(* Schneider Machine Expert - Basic project PICK AND PLACE 1.2mantep, file version 2.7.0.0 *)
(* ProjectInformations: Name=New project *)

HARDWARE
  Cpu 0: TM221CE40R
  EthernetConfiguration: NetworkName=M221, IpAllocationMode=FixedAddress, IpAddress=192.168.0.12, SubnetMask=255.255.255.0
  SerialLineConfiguration: Baud=Baud19200, Parity=ParityEven, DataBits=DataBits8, StopBits=StopBits1, PhysicalMedium=PhysicalMediumRs485, TransmissionMode=TransmissionModeModbusRtu, SlaveId=1, Addressing=SlaveAddressing
  MastTask: UsePeriodScanMode=false, PeriodScan=100
  FastTask: Period=255
  CpuBehavior: StartingMode=StartAsPreviousState, AutoSaveRamOnEeprom=true, WatchdogPeriod=250

SYMBOLS  (address, symbol, comment, settings)
  %M0         "K EMG"
  %M1         "K RESET"
  %M2         "RESET CLEAR"
  %M10        "K AUTO"
  %M11        "K1"
  %M12        "K2"
  %M13        "K3"
  %M14        "K4"
  %M15        "K CYC"
  %M16        "K STOP"
  %M17        "K5"
  %M50        "STEP"
  %M51        "K1 STEP"
  %M52        "K2 STEP"
  %M53        "K3 STEP"
  %M54        "K4 STEP"
  %M57        "K5 STEP"
  %M100       "kAmin"
  %M101       "kAplus"
  %M102       "kBmin"
  %M103       "kBplus"
  %M104       "kVakum"
  %M105       "KLHijau"
  %M106       "kLMerah"
  %M107       "kLKuning"
  %M200       "kB1"
  %M201       "kStart"
  %M202       "kStop"
  %M203       "kReset"
  %M204       "kA/S"
  %M205       "kS/C"
  %M206       "kA0"
  %M207       "kLimitS"
  %M208       "kProxy"
  %M209       "kB1min"
  %M210       "kVakum"
  %M211       "kBplus"
  %M212       "kAmin"
  %M213       "kBmin"
  %M214       "kAplus"
  %M215       "kLrun"
  %M216       "kLstop"
  %M217       "kLReset"
  %M400       "M.koilStart"
  %M500       "M.Start"
  %M501       "M.stop"
  %M510       "Mmasterstart"
  %M511       "R_Trig"
  %M700       "K.start"
  %TM0        [Preset=1, Base=OneSecond]
  %TM1        [Preset=1, Base=OneSecond]
  %I0.0       "EMG"
  %I0.1       "START"
  %I0.2       "STOP"
  %I0.3       "RESET"
  %I0.4       "AUTO/STEP"
  %I0.5       "SGL/CYC"
  %I0.7       "A1"
  %I0.10      "A0"
  %I0.11      "LS"
  %I0.12      "PROXY"
  %I0.13      "B1"
  %I0.14      "B1"
  %Q0.3       "VAKUUM"
  %Q0.4       "B+"
  %Q0.5       "A-"
  %Q0.6       "B-"
  %Q0.7       "A+"
  %Q0.11      "IND RUN"
  %Q0.12      "IND STOP"
  %Q0.15      "IND RESET"

POU EMG
  (* SectionNumber=1 *)

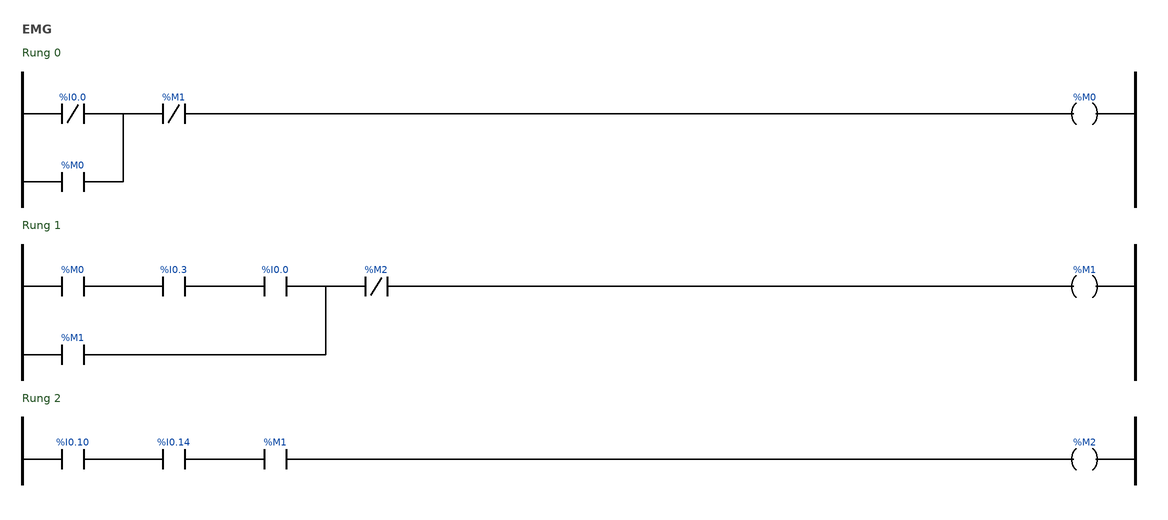

// Rung 0
  LDN %I0.0
  OR %M0
  ANDN %M1
  ST %M0
  // as ST:
  //   %M0 := (NOT %I0.0 OR %M0) AND NOT %M1;

// Rung 1
  LD %M0
  AND %I0.3
  AND %I0.0
  OR %M1
  ANDN %M2
  ST %M1
  // as ST:
  //   %M1 := (%M0 AND %I0.3 AND %I0.0 OR %M1) AND NOT %M2;

// Rung 2
  LD %I0.10
  AND %I0.14
  AND %M1
  ST %M2
  // as ST:
  //   %M2 := %I0.10 AND %I0.14 AND %M1;

POU OUTPUT
  (* SectionNumber=2 *)

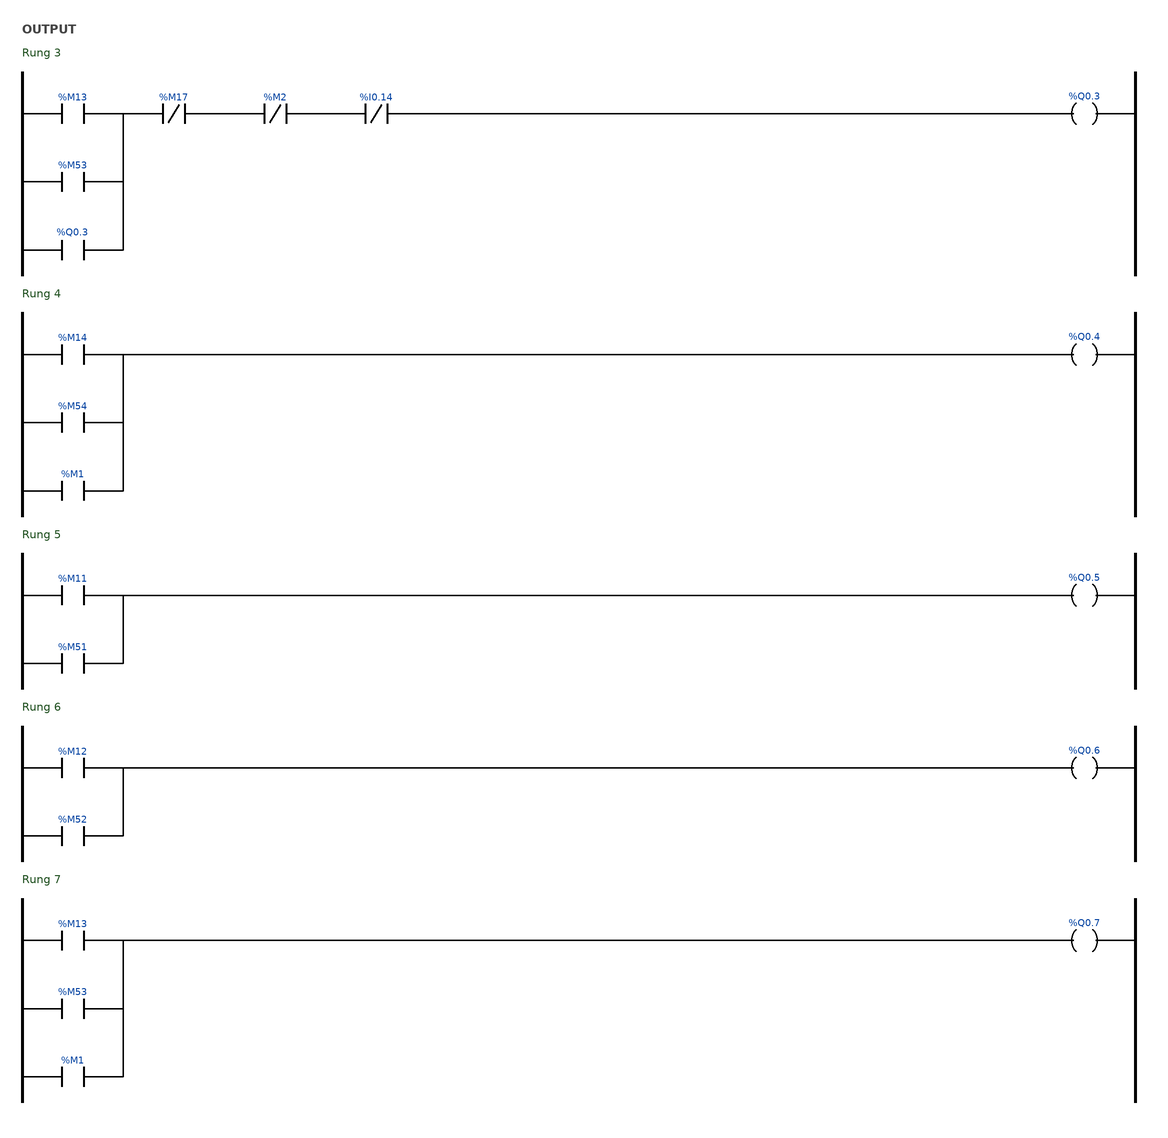

// Rung 3
  LD %M13
  OR %M53
  OR %Q0.3
  ANDN %M17
  ANDN %M2
  ANDN %I0.14
  ST %Q0.3
  // as ST:
  //   %Q0.3 := (%M13 OR %M53 OR %Q0.3) AND NOT %M17 AND NOT %M2 AND NOT %I0.14;

// Rung 4
  LD %M14
  OR %M54
  OR %M1
  ST %Q0.4
  // as ST:
  //   %Q0.4 := %M14 OR %M54 OR %M1;

// Rung 5
  LD %M11
  OR %M51
  ST %Q0.5
  // as ST:
  //   %Q0.5 := %M11 OR %M51;

// Rung 6
  LD %M12
  OR %M52
  ST %Q0.6
  // as ST:
  //   %Q0.6 := %M12 OR %M52;

// Rung 7
  LD %M13
  OR %M53
  OR %M1
  ST %Q0.7
  // as ST:
  //   %Q0.7 := %M13 OR %M53 OR %M1;

POU AUTO
  (* SectionNumber=3 *)

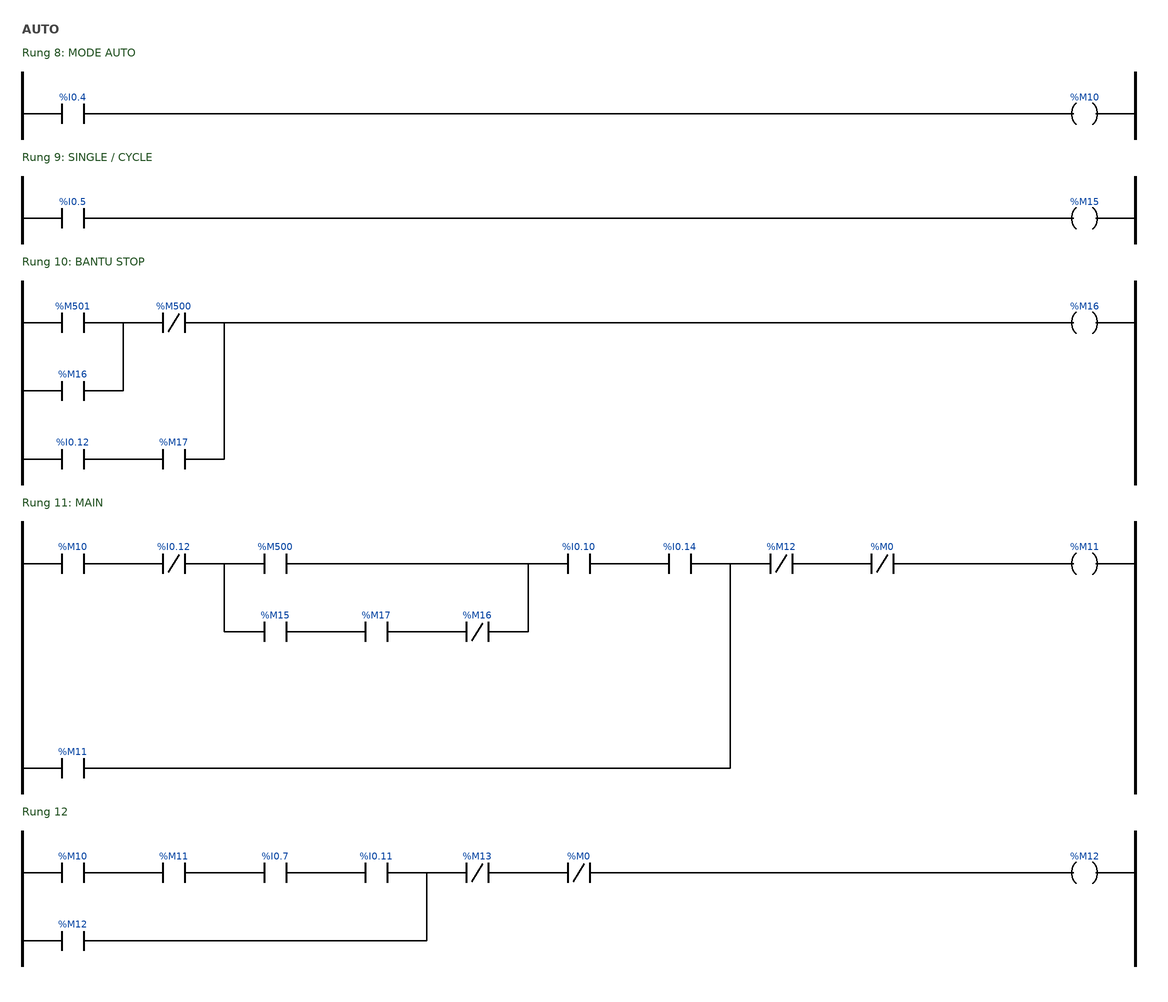

// Rung 8: MODE AUTO
  LD %I0.4
  ST %M10
  // as ST:
  //   %M10 := %I0.4;

// Rung 9: SINGLE / CYCLE
  LD %I0.5
  ST %M15
  // as ST:
  //   %M15 := %I0.5;

// Rung 10: BANTU STOP
  LD %M501
  OR %M16
  ANDN %M500
  OR( %I0.12
  AND %M17
  )
  ST %M16
  // as ST:
  //   %M16 := (%M501 OR %M16) AND NOT %M500 OR %I0.12 AND %M17;

// Rung 11: MAIN
  LD %M10
  ANDN %I0.12
  AND( %M500
  OR( %M15
  AND %M17
  ANDN %M16
  )
  )
  AND %I0.10
  AND %I0.14
  OR %M11
  ANDN %M12
  ANDN %M0
  ST %M11
  // as ST:
  //   %M11 := (%M10 AND NOT %I0.12 AND (%M500 OR %M15 AND %M17 AND NOT %M16) AND %I0.10 AND %I0.14 OR %M11) AND NOT %M12 AND NOT %M0;

// Rung 12
  LD %M10
  AND %M11
  AND %I0.7
  AND %I0.11
  OR %M12
  ANDN %M13
  ANDN %M0
  ST %M12
  // as ST:
  //   %M12 := (%M10 AND %M11 AND %I0.7 AND %I0.11 OR %M12) AND NOT %M13 AND NOT %M0;

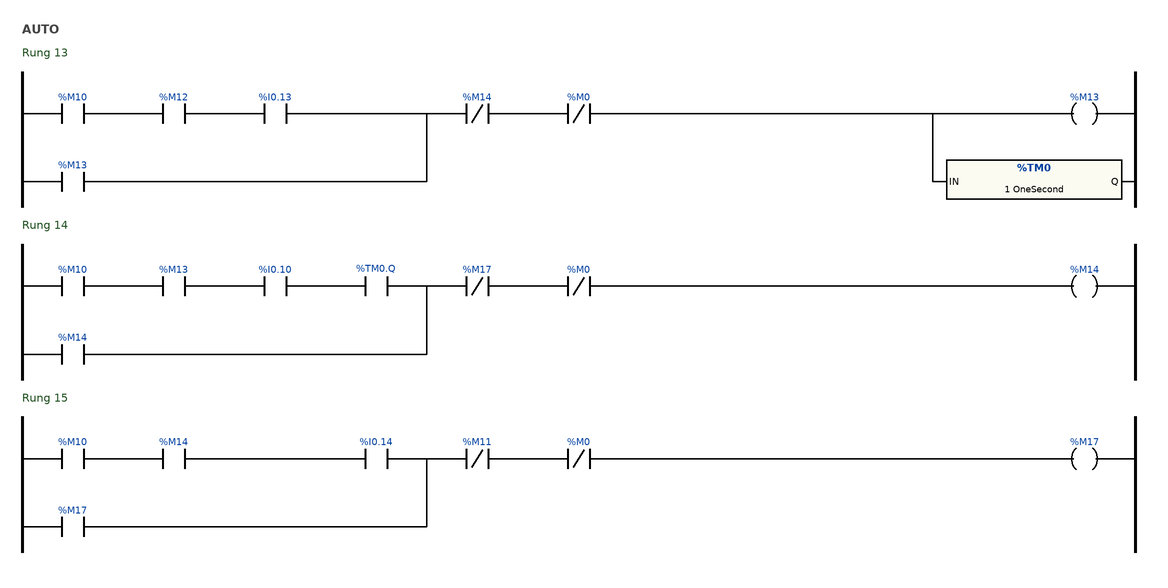

// Rung 13
  LD 1
  MULTIFB
  LD 1
  AND %M10
  AND %M12
  AND %I0.13
  OR %M13
  ANDN %M14
  ANDN %M0
  ST %MW2009:X0
  LD %MW2009:X0
  ST %M13
  BLK %TM0
  LD %MW2009:X0
  IN
  END_BLK
  MULTIFB
  // as ST:
  //   _t1 := (%M10 AND %M12 AND %I0.13 OR %M13) AND NOT %M14 AND NOT %M0;
  //   %M13 := _t1;
  //   %TM0(IN := _t1);

// Rung 14
  LD %M10
  AND %M13
  AND %I0.10
  AND %TM0.Q
  OR %M14
  ANDN %M17
  ANDN %M0
  ST %M14
  // as ST:
  //   %M14 := (%M10 AND %M13 AND %I0.10 AND %TM0.Q OR %M14) AND NOT %M17 AND NOT %M0;

// Rung 15
  LD %M10
  AND %M14
  AND %I0.14
  OR %M17
  ANDN %M11
  ANDN %M0
  ST %M17
  // as ST:
  //   %M17 := (%M10 AND %M14 AND %I0.14 OR %M17) AND NOT %M11 AND NOT %M0;

POU STEP
  (* SectionNumber=4 *)

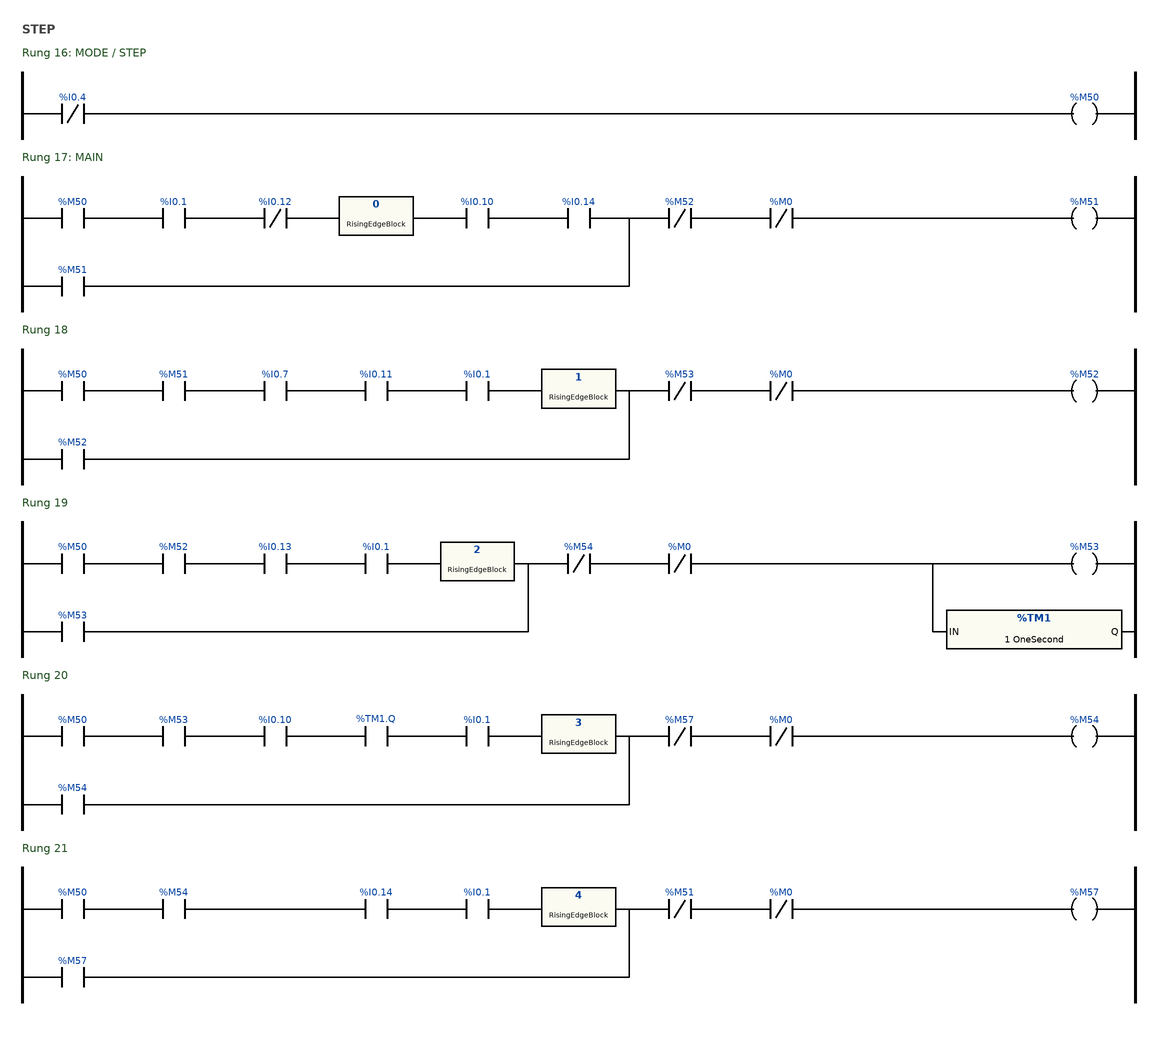

// Rung 16: MODE / STEP
  LDN %I0.4
  ST %M50
  // as ST:
  //   %M50 := NOT %I0.4;

// Rung 17: MAIN
  LD %M50
  AND %I0.1
  ANDN %I0.12
  RISING0
  AND %I0.10
  AND %I0.14
  OR %M51
  ANDN %M52
  ANDN %M0
  ST %M51
  // as ST:
  //   %M51 := (RISING(%M50 AND %I0.1 AND NOT %I0.12) AND %I0.10 AND %I0.14 OR %M51) AND NOT %M52 AND NOT %M0;

// Rung 18
  LD %M50
  AND %M51
  AND %I0.7
  AND %I0.11
  AND %I0.1
  RISING1
  OR %M52
  ANDN %M53
  ANDN %M0
  ST %M52
  // as ST:
  //   %M52 := (RISING(%M50 AND %M51 AND %I0.7 AND %I0.11 AND %I0.1) OR %M52) AND NOT %M53 AND NOT %M0;

// Rung 19
  LD 1
  MULTIFB
  LD 1
  AND %M50
  AND %M52
  AND %I0.13
  AND %I0.1
  RISING2
  OR %M53
  ANDN %M54
  ANDN %M0
  ST %MW2009:X0
  LD %MW2009:X0
  ST %M53
  BLK %TM1
  LD %MW2009:X0
  IN
  END_BLK
  MULTIFB
  // as ST:
  //   _t1 := (RISING(%M50 AND %M52 AND %I0.13 AND %I0.1) OR %M53) AND NOT %M54 AND NOT %M0;
  //   %M53 := _t1;
  //   %TM1(IN := _t1);

// Rung 20
  LD %M50
  AND %M53
  AND %I0.10
  AND %TM1.Q
  AND %I0.1
  RISING3
  OR %M54
  ANDN %M57
  ANDN %M0
  ST %M54
  // as ST:
  //   %M54 := (RISING(%M50 AND %M53 AND %I0.10 AND %TM1.Q AND %I0.1) OR %M54) AND NOT %M57 AND NOT %M0;

// Rung 21
  LD %M50
  AND %M54
  AND %I0.14
  AND %I0.1
  RISING4
  OR %M57
  ANDN %M51
  ANDN %M0
  ST %M57
  // as ST:
  //   %M57 := (RISING(%M50 AND %M54 AND %I0.14 AND %I0.1) OR %M57) AND NOT %M51 AND NOT %M0;

POU Kepserver
  (* SectionNumber=5 *)

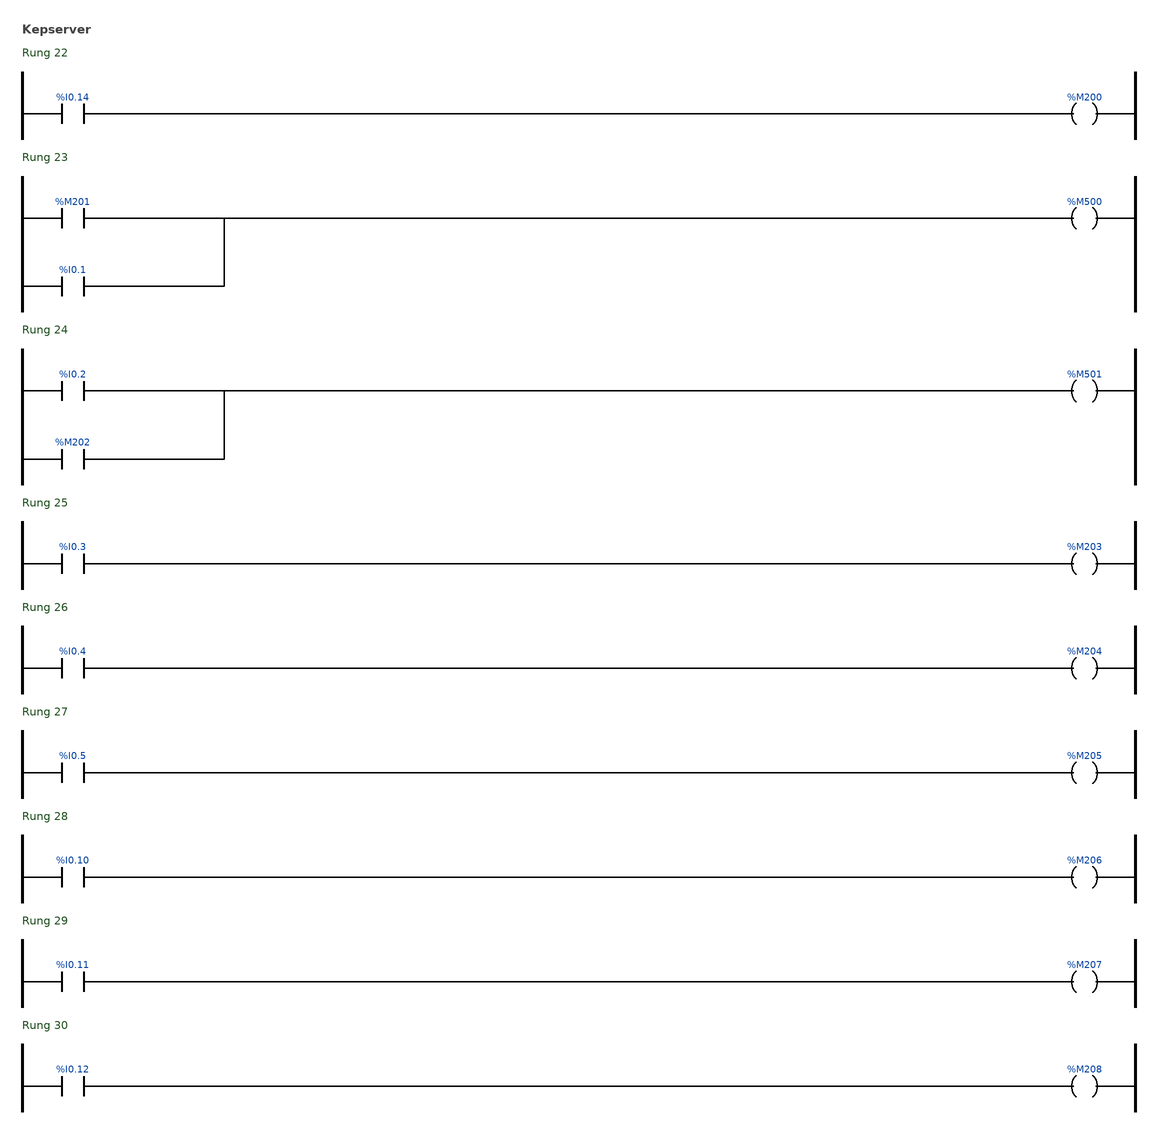

// Rung 22
  LD %I0.14
  ST %M200
  // as ST:
  //   %M200 := %I0.14;

// Rung 23
  LD %M201
  OR %I0.1
  ST %M500
  // as ST:
  //   %M500 := %M201 OR %I0.1;

// Rung 24
  LD %I0.2
  OR %M202
  ST %M501
  // as ST:
  //   %M501 := %I0.2 OR %M202;

// Rung 25
  LD %I0.3
  ST %M203
  // as ST:
  //   %M203 := %I0.3;

// Rung 26
  LD %I0.4
  ST %M204
  // as ST:
  //   %M204 := %I0.4;

// Rung 27
  LD %I0.5
  ST %M205
  // as ST:
  //   %M205 := %I0.5;

// Rung 28
  LD %I0.10
  ST %M206
  // as ST:
  //   %M206 := %I0.10;

// Rung 29
  LD %I0.11
  ST %M207
  // as ST:
  //   %M207 := %I0.11;

// Rung 30
  LD %I0.12
  ST %M208
  // as ST:
  //   %M208 := %I0.12;

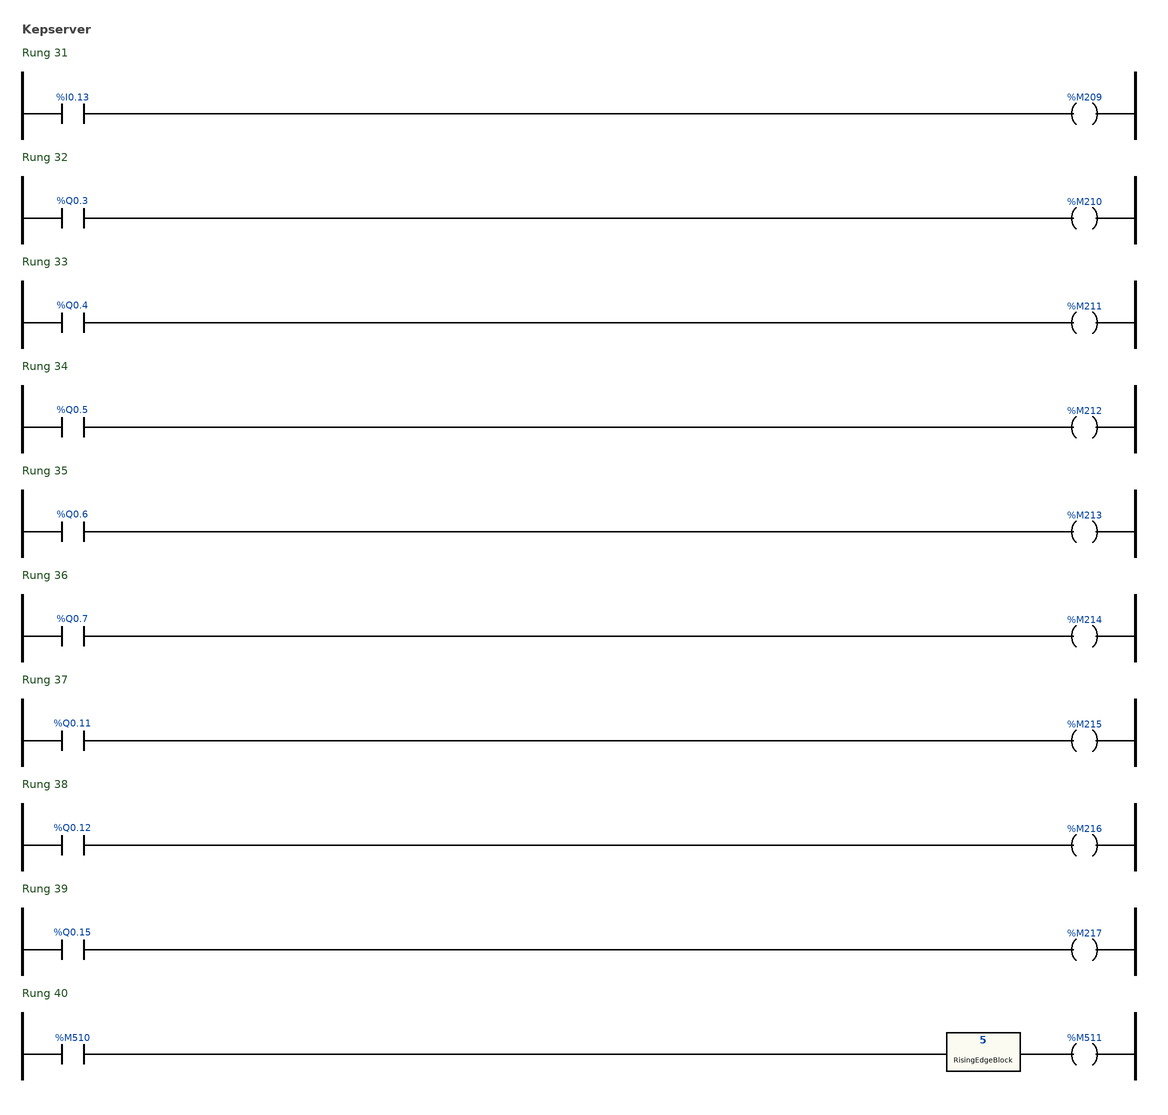

// Rung 31
  LD %I0.13
  ST %M209
  // as ST:
  //   %M209 := %I0.13;

// Rung 32
  LD %Q0.3
  ST %M210
  // as ST:
  //   %M210 := %Q0.3;

// Rung 33
  LD %Q0.4
  ST %M211
  // as ST:
  //   %M211 := %Q0.4;

// Rung 34
  LD %Q0.5
  ST %M212
  // as ST:
  //   %M212 := %Q0.5;

// Rung 35
  LD %Q0.6
  ST %M213
  // as ST:
  //   %M213 := %Q0.6;

// Rung 36
  LD %Q0.7
  ST %M214
  // as ST:
  //   %M214 := %Q0.7;

// Rung 37
  LD %Q0.11
  ST %M215
  // as ST:
  //   %M215 := %Q0.11;

// Rung 38
  LD %Q0.12
  ST %M216
  // as ST:
  //   %M216 := %Q0.12;

// Rung 39
  LD %Q0.15
  ST %M217
  // as ST:
  //   %M217 := %Q0.15;

// Rung 40
  LD %M510
  RISING5
  ST %M511
  // as ST:
  //   %M511 := RISING(%M510);

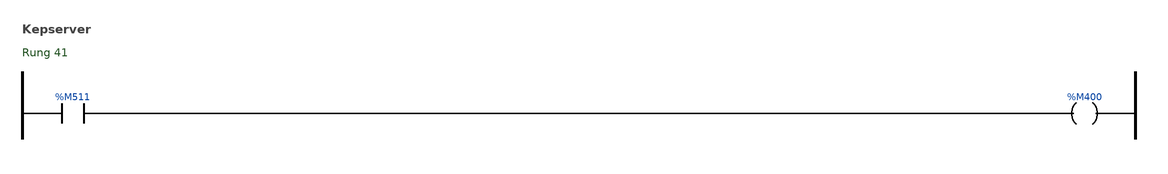

// Rung 41
  LD %M511
  ST %M400
  // as ST:
  //   %M400 := %M511;

POU INDIKATOR
  (* SectionNumber=6 *)

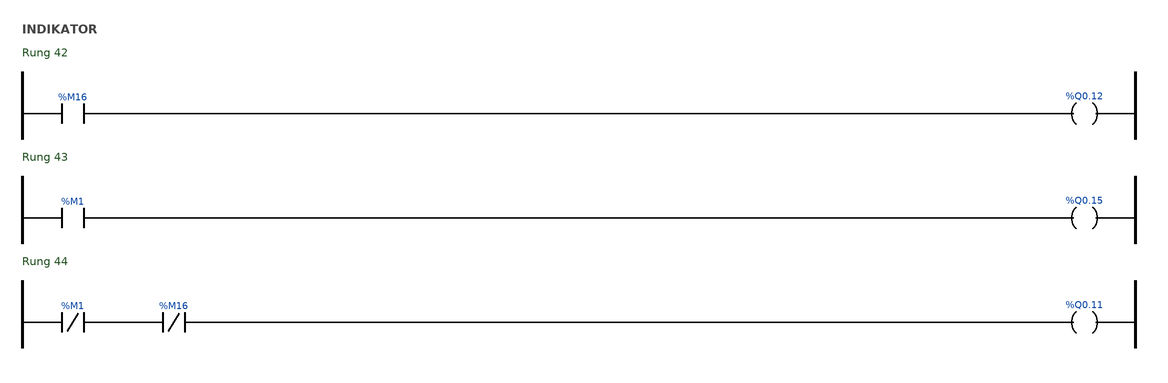

// Rung 42
  LD %M16
  ST %Q0.12
  // as ST:
  //   %Q0.12 := %M16;

// Rung 43
  LD %M1
  ST %Q0.15
  // as ST:
  //   %Q0.15 := %M1;

// Rung 44
  LDN %M1
  ANDN %M16
  ST %Q0.11
  // as ST:
  //   %Q0.11 := NOT %M1 AND NOT %M16;
